TYPE trafficlight_cmds_typ :
STRUCT
	cmdStart:BOOL;
END_STRUCT
END_TYPE

(* stored: Version 1.1.0.1
   DUT trafficlight_cmds_typ: Id {ff8fa796-6080-4a60-8bbf-0db3155f42a5} *)
